# EPICS autosave request: iocBoot/iocTomoScan_BEATS_PCO_ACS_Cont/auto_settings.req
file "tomoScan_settings.req", P=$(P), R=$(R)
file "tomoScan_BEATS_PCO_ACS_Cont_settings.req", P=$(P), R=$(R)
